// TIA Portal V20 export
// export: Created 2025-09-14T11:17:00.0000000Z, ExportSetting WithDefaults
VAR_GLOBAL   // PLC tag table "TagTable_AO"
   RTU1_SF_SpeedRef AT %QW64 : Real;
   RTU1_DMP_PosCmd AT %QW66 : Real;
END_VAR
